INTERFACE I_AxisParameters

PROPERTY AxisParamsError : BOOL
GET
END_GET
END_PROPERTY

PROPERTY AxisParamsErrorID : UDINT
GET
END_GET
END_PROPERTY

PROPERTY AxisParamsInit : BOOL
GET
END_GET
END_PROPERTY

METHOD EncoderParamsSave
VAR_INPUT
    Enable : BOOL;
END_VAR
END_METHOD

METHOD ExposeAxisParams
VAR_INPUT
    Enable: BOOL;
    RefreshDelay: TIME;
END_VAR
END_METHOD

PROPERTY RefVeloSearch : LREAL
GET
END_GET
END_PROPERTY

PROPERTY RefVeloSync : LREAL
GET
END_GET
END_PROPERTY

METHOD RestoreAxisParams
VAR_INPUT
END_VAR
END_METHOD

PROPERTY RestoreDone : BOOL
GET
END_GET
END_PROPERTY

PROPERTY SavedPosition : LREAL
GET
END_GET
END_PROPERTY

PROPERTY ScaledEncoderCount : UDINT
GET
END_GET
END_PROPERTY

METHOD ScaleRawEncoder : UDINT
END_METHOD

END_INTERFACE

(* stored: Version 1.1.0.1
   Itf I_AxisParameters: Id {f91fa392-42b9-4cf5-a843-28456ed2820b}
   Property AxisParamsError: Id {e9e077a6-6930-4649-85af-c395ca806531}
   Get Get: Id {a63dffe9-b0a4-48a7-a237-0a9129339422}
   Property AxisParamsErrorID: Id {0f4330bf-83b2-422b-8828-706ab87543cd}
   Get Get: Id {9780000b-60a0-4a5c-8cf0-365a7339a4b4}
   Property AxisParamsInit: Id {0aff11b7-df26-41a4-b267-6edbd4c57328}
   Get Get: Id {79d5f5f5-86e1-4e26-b4c1-b2fd6f35a037}
   Method EncoderParamsSave: Id {543b2f95-a551-4fd8-9961-1f96cda4fa13}
   Method ExposeAxisParams: Id {4789401e-3661-49e3-b98c-e95d7eff7616}
   Property RefVeloSearch: Id {8a35fa96-dbfb-404d-93a0-e871a2d3d063}
   Get Get: Id {e8cf9088-9695-42fc-8b81-7f13211fe1dc}
   Property RefVeloSync: Id {a25eef31-589e-4b83-ab70-cb029abd6e98}
   Get Get: Id {10344ee7-2ae2-48ac-9706-25700bcdf13f}
   Method RestoreAxisParams: Id {507dd76e-711b-4765-ae75-25397b03046b}
   Property RestoreDone: Id {6c7c316a-24ab-45a6-b98f-53642b5389c7}
   Get Get: Id {8b50b761-13ce-41f8-8f76-0dd608718848}
   Property SavedPosition: Id {3eb2be5e-1bc5-4267-9504-fd4efa432df8}
   Get Get: Id {3d3eebab-1130-4c6e-a759-bbdd38ce8881}
   Property ScaledEncoderCount: Id {93445dbc-b389-4916-96fe-856216773594}
   Get Get: Id {34af533c-cf5f-4a77-a012-16b3af7602a0}
   Method ScaleRawEncoder: Id {aa4aa2b3-d892-434a-940d-c34b50da3016} *)
